// TIA Portal V20 export
// export: Created 2025-12-01T14:56:21.9472908Z, ExportSetting None, DisplayName Totally Integrated Automation Portal, DisplayVersion V20 Update 3, DisplayName TIA Portal Openness, DisplayVersion V20 Update 3, DisplayName TIA Portal Version Control Interface, DisplayVersion V20 Update 3, DisplayName STEP 7 Professional, DisplayVersion V20 Update 3, DisplayName STEP 7 Safety, DisplayVersion V20 Update 2, DisplayName WinCC Basic/Comfort/Advanced, DisplayVersion V20 Update 3, DisplayName WinCC Professional, DisplayVersion V20 Update 3, DisplayName WinCC Unified, DisplayVersion V20 Update 3
TYPE "CBS_Datos_config"
   STRUCT
      Numero_MesaAsociada : UInt;   // Numero de Mesa Asociado al Quimarox
      Numero_vagones : Int;
      ConfigEvento : Struct
         SSCC : Bool;
      END_STRUCT;
      Long_Vagon_mm : Int;
      Long_Util_vagon_mm : Int;
      dist_ini_vag_a_phs_mm : Int;
      maximo_encoder : DInt;
      relacion_mm_pulso : Real;
      DatosTrabajo : Struct
         Memoria_Dato_Encoder : DInt;
         Hora_Ultimo_Refresco : Time_Of_Day;
         Hora_Anterior_Refresco : Time_Of_Day;
         Memoria_MCKEY : UDInt;
         Actualizar_Config : Bool;
         Memoria_Inicializacion : Bool;
         Memoria_Actualizacion_Config : Bool;
         Error_Referenciacion : Bool;
         Error_Timeout_Com_SAC : Bool;
      END_STRUCT;
   END_STRUCT;
END_TYPE
